(* IEC 61131-3 sources: com.logicals.lc3.webinar/RPMControl_Webinar/src_PRG_MQTT_RevPi_ST, 4 files *)

(* ---- PRG_RevPi_MQTTConnect.iecst ---- *)
/*
 * TauriL
 * MQTTConnect Task
 */

USING com.logicals.Basic.Logic;

PROGRAM PRG_RevPi_MQTTConnect

    VAR_EXTERNAL
      gstruc_MQTTClient    : DT_MQTTClient;
    END_VAR

    VAR_EXTERNAL
      /*
       * Funktion Publish starten (WebCon)
       */
       gx_MQTTPublish      : BOOL;
       gx_MQTTPublishState : BOOL;
    END_VAR

    VAR_EXTERNAL
       /*
        * Funktion Subscribe starten (WebCon)
        */
        gx_MQTTSubscribe      : BOOL;
        gx_MQTTSubscribeState : BOOL;
    END_VAR

   /*
    * PRG_RevPi_MQTTConnect
    */
	VAR_EXTERNAL
      /*
       * Globaler TraceLevel
       */
       gui_TraceLevel : UINT;
	END_VAR
   /*
    * Status Verbindung zum Broker
    */
	VAR_EXTERNAL
		/*
		 * State und Channel vom Connect
		 */
		 MQTT_State   : MQTT_SUBSCRIBER_STATE;
		 MQTT_Channel : DINT;
	END_VAR

    VAR_EXTERNAL
        /*
         * Conecting Status an WebCon
         */
         gui_MQTTConnecting    : UINT; // Anzahl der Zyklen in MQTTConnecting
        /*
         * Conect und DisConnect Status an WebCon
         */
	     gui_MQTTConOkCycle    : UINT; // Anzahl der Zyklen bis MQTT Connect
	     gui_MQTTConNotOkCycle : UINT; // Anzahl der Zyklen wenn MQTT DisConnect
        /*
         * Conect Status an WebCon
         */
         gx_MQTTConOk      : BOOL;
    END_VAR

    VAR

    l_ConState : MQTT_SUBSCRIBER_STATE;

    l_RC       : MQTT_RC;
    ldi_Ch     : DINT;

    l_RC_Disconnect : MQTT_RC;

  END_VAR

   VAR
    /*
     * DiagnoseBits fuer RTS
     */
     lx_RTSInit     : BOOL;
     lx_RTSRun      : BOOL;
     lx_RTSShutDown : BOOL;
     lx_RTSTerm     : BOOL;
   END_VAR

   VAR
	 //
	 // Aus HCLib
     // Alle Verbindungen bedienen
     // Hier werden die Daten konkret verschickt!
     FB_RevPi_MQTTConnect        : FB_MQTTConnect;
  END_VAR

 /*
  * Status MQTT Publish/Subscribe
  */
  VAR
     FB_Publish_Toogle         : FB_lc_Toggle_ST;
     FB_Subscribe_Toogle       : FB_lc_Toggle_ST;
  END_VAR

  VAR
    FB_MQTTCpyRevPiPar : FB_MQTTCpyRevPiPar;
  END_VAR

  VAR
    /*
     * Der Datentyp enthaelt alle wesentlichen Informationen f�r die Basis-
     * Einstellungen von MQTT
     */
     l_MQTTInitKom    : DT_MQTT;
  END_VAR

 /*
  * Initialisierungsmerker
  */
  VAR
     FB_InitR_TRIG       : R_TRIG;
  END_VAR

  VAR
    /* Lokaler InitPuls im Baustein */
     lx_CycleInit : BOOL;

    /* Lokaler Puls im Baustein */
     lx_CyclePulse : BOOL;
    /* Lokaler Zyklustaktzaehler */
     li_CycleCount : INT;

    /* Lokaler InitZyklustaktzaehler */
     li_CycleCountInitVal : INT;
  END_VAR

  VAR
    lstr_PRGName      : STRING[30] := 'PRG_RevPi_MQTTConnect';
    lui_TraceLevel    : UINT     := 5;

    lui_POU_UID       : UINT;                                      // Lokale POU-ID
    lstr_InstName     : STRING[30];
    lstr_POU_InstPath : STRING[128];                               // Lokale POU-ID
   END_VAR
 /*
  * -------------------------------------------------
  * Start SPS-Programm PRG_RevPi_MQTTConnect
  * -------------------------------------------------
  */
 /*
  * InitZyklus setzen wenn MQTT aktiv gesetzt!
  */
  FB_InitR_TRIG(CLK := TRUE,Q => lx_CycleInit);

 /*
  * CyclePulse
  */
  lx_CyclePulse := NOT(lx_CyclePulse);

 /*
  * LifeTick bzw. ZyklusZaehler
  */
  li_CycleCount := li_CycleCount + 1;

  IF lx_CycleInit = TRUE THEN
       /*
        * Globalen TraceLevel uebernehmen
        */
       lui_TraceLevel := gui_TraceLevel;
      /*
       * PI-Name fuer GVL-Liste
       */
       lstr_InstName        := GET_CURRENT_PI_NAME();
       lstr_POU_InstPath    := lstr_PRGName;
       li_CycleCountInitVal := li_CycleCountInitVal + 1;
   END_IF;

  /*
   * MQTT Parameter umkopieren
   */
   IF lx_CycleInit = TRUE THEN
    FB_MQTTCpyRevPiPar(vistruc_InitKom := l_MQTTInitKom,
                       vostruc_InitKom => gstruc_MQTTClient);
   END_IF;

   /*
    * Betriebsart MQTT von Visu
    * Publish der Daten immer aus TRUE im CycleInit setzen
    */
    FB_Publish_Toogle(vix_In := gx_MQTTPublish OR lx_CycleInit,vox_Out => gx_MQTTPublishState);
    FB_Subscribe_Toogle(vix_IN := gx_MQTTSubscribe, vox_Out =>gx_MQTTSubscribeState);

    /*
     * Es wird ein MQTT_Connect aufgebaut
     * Wird fuer Publish/Subscribe verwendet!
     * NUR ein Connect je Resource zum Broker erlaubt!
     *
     * Im RTSTerm bzw. RTSShutdown MUSS der Connect Disconnected werden!
     */
     FB_RevPi_MQTTConnect(vistr_InstPath                := lstr_InstName,
     	                  vistr_BrokerAddress          := l_MQTTInitKom.BrokerAdress,
                          vistr_ClientID               := l_MQTTInitKom.RevPiClientID,
                          vo_State                     => l_ConState,              // Status fuer Connect fuer alle zu oeffnenden Verbindungen (Pub/Sub) zum Broker
                          vo_RC                        => l_RC,                    // Status fuer Connect fuer alle zu oeffnenden Fehler (Pub/Sub) zum Broker
                          vodi_ch                      => ldi_Ch,                  // Status fuer Connect fuer alle zu oeffnenden Kanaele (Pub/Sub) zum Broker
                          voui_CycleCount_Connecting   => gui_MQTTConnecting,
                          voui_CycleCount_Connected    => gui_MQTTConOkCycle,      // Wert auch in WebCon
                          voui_CycleCount_NotConnected => gui_MQTTConNotOkCycle,   // Wert auch in WebCon
                          vox_MQTTConOk                => gx_MQTTConOk);           // Wert auch in WebCon

   gstruc_MQTTClient.x_MQTTConOk          := gx_MQTTConOk;
   gstruc_MQTTClient.ui_MQTTConnecting    := gui_MQTTConnecting;
   gstruc_MQTTClient.ui_MQTTConOkCycle    := gui_MQTTConOkCycle;
   gstruc_MQTTClient.ui_MQTTConNotOkCycle := gui_MQTTConNotOkCycle;

   /*
    * Ausgabe der Daten!
    */
    MQTT_State   := l_ConState;
    MQTT_Channel := ldi_ch;

   /*
    * Diagnosebits des RTS
    */
    RTSCycleInfo(Init     => lx_RTSInit,
  	             Run      => lx_RTSRun,
  	             Shutdown => lx_RTSShutDown,
  	             Term     => lx_RTSTerm);

   /*
    * Disconnect!
    * In RTS.CFG ShutDown Cycle von 3 Sekunden eintragen!
    */
    IF lx_RTSTerm = TRUE OR lx_RTSShutDown = TRUE THEN
     MQTT_Disconnect(ch := ldi_ch,
                     rc => l_RC_Disconnect);
     MQTT_State   := l_ConState;
     MQTT_Channel := -1;
    END_IF;

END_PROGRAM

(* ---- PRG_RevPi_MQTTPublish_Header.iecst ---- *)
 /*
  * logi.cals GmbH
  * A-3100 St. Poelten
  * Europaplatz 7/1
  * Tel.: 0043-5-77147
  *
  * logi.cals automation solutions & services GmbH
  * D-40738 Langenfeld
  * Postfach 1306
  * Tel.: 0043-5-77147
  *
  * Contact:
  * dieter.goltz@logicals.com
  *
  * History:
  * Created:
  * DG 2021-05-30 MQTT Header
  *
  * Modified:
  * DG 2021-05-30 MQTT Publish Header
  */

 /*
  * Description
  * ===========
  */

 /*
  * Beschreibung
  * ============
  * MQTT Kommunikation
  * Publish Header
  *
  */

/*
 * Lokaler Test
 * ============
 * sudo mosquitto_sub -d -t test   - test = Name des Topic -> /Tauri       - Header
 *                                                            /Tauri       - Werte
 *
 * sudo mosquitto_pub -d -t test –m “Hello” - test = Name des Topic -> /GHaus       - Header
 *                                                                     /GHaus/Value - Werte
 *
 *                               -m "Hello" -> String der verschickt wird!
 */

/*
 * Publish des Header von TauriL
 */
PROGRAM PRG_RevPi_MQTTPublish_Header
    /*
	 * PRG_RevPi_MQTTPublish_Header
	 */
    VAR_EXTERNAL
         MQTTHeader       : MQTTHeader;
    END_VAR

    VAR_EXTERNAL
        /*
         * Funktion Publish starten (WebCon)
         * Wird in MQTTConnect gesetzt!
         * Kann von hier mit gx_MQTTPublish getoggled werden!
         */
         gx_MQTTPublish      : BOOL;
         gx_MQTTPublishState : BOOL;
    END_VAR

	VAR_EXTERNAL
	   /*
		* State und Channel vom Connect
		*/
		MQTT_State   : MQTT_SUBSCRIBER_STATE;
		MQTT_Channel : DINT;
	END_VAR

	VAR_EXTERNAL
      /*
       * Globaler TraceLevel
       */
     gui_TraceLevel : UINT;
	END_VAR

	VAR_EXTERNAL
    /*
     * Uhrzeit und Daten von TimeBaustein abholen
     * und auf Globale Var in Byte schreiben
     * Fuer MQTT
     */
  	 gb_RTSSeconds : BYTE;
 	 gb_RTSMinutes : BYTE;
	 gb_RTSHours   : BYTE;

	 gb_RTSDay         : BYTE;
	 gb_RTSMonth       : BYTE;
	 gb_RTSYearHByte   : BYTE;
	 gb_RTSYearLByte   : BYTE;

    END_VAR

   VAR
      FB_MQTT_PublishRevPi      : FB_MQTT_Publish;
   END_VAR

  VAR
    /*
     * Der Datentyp enthaelt alle wesentlichen Initwerte f�r die MQTT-Kommunkation
     */
     l_MQTTInitKom         : DT_MQTT;
    /*
     * Status-Informationen
     */
     ldi_PublishLifeTick : DINT;
     lx_PublishOK        : BOOL;
     lui_IPVal1          : UINT;
     lui_IPVal2          : UINT;
     lui_IPVal3          : UINT;
     ldint_MQTTChannel   : DINT;
     ldint_MQTTCount     : DINT;
     ldint_MQTTrc        : DINT;
     lsint_MQTTState     : SINT;
     lx_MQTTENO          : BOOL;
     luint_MQTTLength    : UINT;
     lui_PubTick         : UINT;
  END_VAR

  VAR
    l_ConState : MQTT_SUBSCRIBER_STATE;
    ldi_ConCh  : DINT;
  END_VAR

  VAR
    lstr_PRGName   : STRING[30] := 'PRG_RevPi_MQTTPublish_Header';
    lui_TraceLevel : UINT     := 5;
  END_VAR

  VAR
     FB_InitR_TRIG       : R_TRIG;
  END_VAR

  VAR
    /* Lokaler InitPuls im Baustein */
     lx_CycleInit : BOOL;

    /* Lokaler Puls im Baustein */
     lx_CyclePulse : BOOL;
    /* Lokaler Zyklustaktzaehler */
     li_CycleCount : INT;

    /* Lokaler InitZyklustaktzaehler */
     li_CycleCountInitVal : INT;
  END_VAR

 /*
  * InitZyklus setzen wenn MQTT aktiv gesetzt!
  */
  FB_InitR_TRIG(CLK := TRUE,Q => lx_CycleInit);
 /*
  * CyclePulse
  */
  lx_CyclePulse := NOT(lx_CyclePulse);

 /*
  * LifeTick bzw. ZyklusZaehler
  */
  li_CycleCount := li_CycleCount + 1;

  /*
   * Steuerung Publish / Subscribe ueber die Visu
   *
   * Publish
   * Welche Daten sollen an den Broker zurueckgeschickt werden
   * Subscribe
   * Welche Daten sollen geholt werden?
   */
   IF lx_CycleInit = TRUE THEN
      /*
       * Init Messages senden
       */
       lui_TraceLevel := gui_TraceLevel;
       li_CycleCountInitVal := li_CycleCountInitVal + 1;
   END_IF;
   /*
    * Daten von MQTTConnect
    */
    l_ConState := MQTT_State;
    ldi_ConCh  := MQTT_Channel;

    IF l_ConState = MQTT_SUBSCRIBER_STATE#CONNECTED THEN

       IF gx_MQTTPublishState = TRUE THEN

     	 MQTTHeader.Second    := gb_RTSSeconds;
   	     MQTTHeader.Minute    := gb_RTSMinutes;
  	     MQTTHeader.Hour      := gb_RTSHours;

  	     MQTTHeader.Day       := gb_RTSDay;
  	     MQTTHeader.Month     := gb_RTSMonth;
  	     MQTTHeader.YearHByte := gb_RTSYearHByte;
  	     MQTTHeader.YearLByte := gb_RTSYearLByte;

         MQTTHeader.IPVal3 := TO_BYTE(RIGHT(IN:= l_MQTTInitKom.RevPiIPAdress, L := 1));
         MQTTHeader.IPVal2 := TO_BYTE(LEFT(RIGHT(IN:= l_MQTTInitKom.RevPiIPAdress, L := 2),1));
         MQTTHeader.IPVal1 := TO_BYTE(LEFT(RIGHT(IN:= l_MQTTInitKom.RevPiIPAdress, L := 3),1));

         FB_MQTT_PublishRevPi(vi_MQTTHeader            := MQTTHeader,
                              vistr_IPAddr             := l_MQTTInitKom.RevPiIPAdress,
                              vistr_BrokerIPAddr       := l_MQTTInitKom.BrokerAdress,
                              vix_Init                 := lx_CycleInit,
                              vi_State                 := l_ConState,
                              vdi_ch                   := ldi_ConCh,
         	                  vistr_BrokerPublishTopic := l_MQTTInitKom.RevPiTopic,
                              vodi_PublishLifeTick     => ldi_PublishLifeTick,
                              vox_PublishOK            => lx_PublishOK,
                              voui_IPVal1              => lui_IPVal1,
                              voui_IPVal2              => lui_IPVal2,
                              voui_IPVal3              => lui_IPVal3,
                              vodint_MQTTChannel       => ldint_MQTTChannel,
                              vodint_MQTTCount         => ldint_MQTTCount,
                              vodint_MQTTrc            => ldint_MQTTrc,
                              vosint_MQTTState         => lsint_MQTTState,
                              vox_MQTTENO              => lx_MQTTENO,
                              vouint_MQTTLength        => luint_MQTTLength,
                              voui_PubTick             => lui_PubTick);

        END_IF;
     END_IF;
END_PROGRAM

(* ---- PRG_RevPi_MQTTPublish_IO.iecst ---- *)
   /*
  * logi.cals GmbH
  * A-3100 St. Poelten
  * Europaplatz 7/1
  * Tel.: 0043-5-77147
  *
  * logi.cals automation solutions & services GmbH
  * D-40738 Langenfeld
  * Postfach 1306
  * Tel.: 0043-5-77147
  *
  * Contact:
  * dieter.goltz@logicals.com
  *
  * History:
  * Created:
  * DG 2021-05-30
  *
  * Modified:
  * DG 2021-05-30 IO
  */

 /*
  * Description
  * ===========
  */

 /*
  * Beschreibung
  * ============
  * MQTT Kommunikation
  * Publish Werte als Topics (IO)
  *
  * Austausch der aktuellen Daten mit dem Broker
  *
  */
 PROGRAM PRG_RevPi_MQTTPublish_IO

   VAR_EXTERNAL
        /*
         * Funktion Publish starten (WebCon)
         */
         gx_MQTTPublish      : BOOL;
         gx_MQTTPublishState : BOOL;
   END_VAR

   VAR_EXTERNAL
	    /* ProcessValue - Analogeingang_1 0..32767 unskaliert */
		gr_PV : REAL;
	    /* SetPoint     - Analogeingang_2 0..32767 unskaliert */
		gr_SP : REAL;
	    /* OutValue     - Analogausgang_1 0..32767 skaliert von 0..100% */
		gr_Y : REAL;
	    /* OutValue     - Ausgang Regler 0..100% wird skaliert auf 0..32767 */
		gr_PID_OUT : REAL;

	    /* ManualWert 0..100% */
		gr_Manual : REAL;

	    /* ProcessValue - Analogeingang_1 Skaliert 0..100%*/
		gr_PV_Scale : REAL;
	    /* SetPoint     - Analogeingang_2 Skaliert 0..100% */
		gr_SP_Scale : REAL;
	    /* OutValue     - Analogausgang_1 Skaliert 0..100% */
		gr_Y_Scale  : REAL;
        /*
         * Anzeige der Betriebsart 1Aus4
         */
        /* An Ausgang Ausgangswert = 0% */
        gx_ModeRPM0 : BOOL;
        /* An Ausgang Ausgangswert = 25% */
        gx_ModeRPM1 : BOOL;
        /* An Ausgang Ausgangswert = 50% */
        gx_ModeRPM2 : BOOL;
        /* An Ausgang SetPoint von Poti */
        gx_ModeRPM3 : BOOL;
        /* An Ausgang SetPoint von SFC */
        gx_ModeRPM4 : BOOL;

        /* Blinkfunktion */
        gx_Flash : BOOL;
   END_VAR
  /*
   * PRG_TauriL_MQTTPublish_IO
   */
   VAR_EXTERNAL
    /*
     * State und Channel vom Connect
     */
     MQTT_State   : MQTT_SUBSCRIBER_STATE;
     MQTT_Channel : DINT;
   END_VAR

   VAR_EXTERNAL
      /*
       * Globaler TraceLevel
       */
       gui_TraceLevel : UINT;
   END_VAR

  /*
   * Publish Topic / BOOL-Status von Topic
   */
   VAR
       FB_MQTT_Publish_IOBlink             : FB_MQTT_Publish_IO;

       FB_MQTT_Publish_IOValModeRPM0       : FB_MQTT_Publish_IO;
       FB_MQTT_Publish_IOValModeRPM1       : FB_MQTT_Publish_IO;
       FB_MQTT_Publish_IOValModeRPM2       : FB_MQTT_Publish_IO;
       FB_MQTT_Publish_IOValModeRPM3       : FB_MQTT_Publish_IO;
       FB_MQTT_Publish_IOValModeRPM4       : FB_MQTT_Publish_IO;

       FB_MQTT_Publish_IOValPV             : FB_MQTT_Publish_IOVal;
       FB_MQTT_Publish_IOValSP             : FB_MQTT_Publish_IOVal;
       FB_MQTT_Publish_IOValY              : FB_MQTT_Publish_IOVal;
       FB_MQTT_Publish_IOValManual         : FB_MQTT_Publish_IOVal;
       FB_MQTT_Publish_IOValPV_Scale       : FB_MQTT_Publish_IOVal;
       FB_MQTT_Publish_IOValSP_Scale       : FB_MQTT_Publish_IOVal;
       FB_MQTT_Publish_IOValY_Scale        : FB_MQTT_Publish_IOVal;

   END_VAR

  VAR
    /*
     * Der Datentyp enthaelt alle wesentlichen Informationen fuer die Basis-
     * Einstellungen von MQTT
     */
     l_MQTTInitKom    : DT_MQTT;
  END_VAR

  VAR
    l_ConState : MQTT_SUBSCRIBER_STATE;
    ldi_ConCh  : DINT;
  END_VAR

   VAR
    lstr_PRGName : STRING[30] := 'PRG_TauriL_MQTTPublish_IO';
    lui_TraceLevel : UINT     := 5;
   END_VAR
 /*
  * Initialisierungsmerker
  */
  VAR
     FB_InitR_TRIG       : R_TRIG;
  END_VAR

  VAR
    /* Lokaler InitPuls im Baustein */
     lx_CycleInit        : BOOL;

    /* Lokaler Puls im Baustein */
     lx_CyclePulse       : BOOL;
    /* Lokaler Zyklustaktzaehler */
     li_CycleCount       : INT;

    /* Lokaler InitZyklustaktzaehler */
     li_CycleCountInitVal : INT;
  END_VAR

  /*
   * InitZyklus setzen wenn MQTT aktiv gesetzt!
   */
   FB_InitR_TRIG(CLK := TRUE,Q => lx_CycleInit);

   lui_TraceLevel := gui_TraceLevel;

  /*
   * CyclePulse
   */
   lx_CyclePulse := NOT(lx_CyclePulse);

  /*
   * LifeTick bzw. ZyklusZaehler
   */
   li_CycleCount := li_CycleCount + 1;
  /*
   * -------------------------------------------------
   * Start SPS-Programm PRG_TauriL_MQTTPublish_IO
   * -------------------------------------------------
   */

  /*
   * Steuerung Publish_IO
   *
   * Publish
   * Welche Einzel-Daten sollen an den Broker geschickt werden
   */
   IF lx_CycleInit = TRUE THEN
       li_CycleCountInitVal := li_CycleCountInitVal + 1;
   END_IF;

   /*
    * Daten von MQTTConnect
    */
    l_ConState := MQTT_State;
    ldi_ConCh  := MQTT_Channel;

   /*
    * Kommt von MQTTConnect
    * Wert MUSS 6 sein!
    */
    IF l_ConState = MQTT_SUBSCRIBER_STATE#CONNECTED /* connected */ THEN

      IF gx_MQTTPublishState = TRUE THEN

      /*
       * Blinkfunktion an gx_Out8
       */
       FB_MQTT_Publish_IOBlink(viui_TraceLevel            := lui_TraceLevel,
                               vix_PubIn                  := gx_Flash,
                               vistr_BrokerPublishTopicIO := l_MQTTInitKom.TauriLTopicIOBlink,
                               vi_State                   := l_ConState,
                               vidi_Ch                    := ldi_ConCh);

      /*
       * Mode RPM 0
       */
       FB_MQTT_Publish_IOValModeRPM0(viui_TraceLevel            := lui_TraceLevel,
                                     vix_PubIn                  := gx_ModeRPM0,
                                     vistr_BrokerPublishTopicIO := l_MQTTInitKom.TauriLTopicIOModeRPM0,
                                     vi_State                   := l_ConState,
                                     vidi_Ch                    := ldi_ConCh);

      /*
       * Mode RPM 1
       */
       FB_MQTT_Publish_IOValModeRPM1(viui_TraceLevel            := lui_TraceLevel,
                                     vix_PubIn                  := gx_ModeRPM1,
                                     vistr_BrokerPublishTopicIO := l_MQTTInitKom.TauriLTopicIOModeRPM1,
                                     vi_State                   := l_ConState,
                                     vidi_Ch                    := ldi_ConCh);

      /*
       * Mode RPM 2
       */
       FB_MQTT_Publish_IOValModeRPM2(viui_TraceLevel            := lui_TraceLevel,
                                     vix_PubIn                  := gx_ModeRPM2,
                                     vistr_BrokerPublishTopicIO := l_MQTTInitKom.TauriLTopicIOModeRPM2,
                                     vi_State                   := l_ConState,
                                     vidi_Ch                    := ldi_ConCh);

      /*
       * Mode RPM 3
       */
       FB_MQTT_Publish_IOValModeRPM3(viui_TraceLevel            := lui_TraceLevel,
                                     vix_PubIn                  := gx_ModeRPM3,
                                     vistr_BrokerPublishTopicIO := l_MQTTInitKom.TauriLTopicIOModeRPM3,
                                     vi_State                   := l_ConState,
                                     vidi_Ch                    := ldi_ConCh);
      /*
       * Mode RPM 4
       */
       FB_MQTT_Publish_IOValModeRPM4(viui_TraceLevel            := lui_TraceLevel,
                                     vix_PubIn                  := gx_ModeRPM4,
                                     vistr_BrokerPublishTopicIO := l_MQTTInitKom.TauriLTopicIOModeRPM4,
                                     vi_State                   := l_ConState,
                                     vidi_Ch                    := ldi_ConCh);
      /*
       * PV
       */
       FB_MQTT_Publish_IOValPV(viui_TraceLevel            := lui_TraceLevel,
                               vir_PubIn                  := gr_PV,
                               vistr_BrokerPublishTopicIO := l_MQTTInitKom.TauriLTopicIOPV,
                               vi_State                   := l_ConState,
                               vidi_Ch                    := ldi_ConCh);

      /*
       * SP
       */
       FB_MQTT_Publish_IOValSP(viui_TraceLevel            := lui_TraceLevel,
                               vir_PubIn                  := gr_SP,
                               vistr_BrokerPublishTopicIO := l_MQTTInitKom.TauriLTopicIOSP,
                               vi_State                   := l_ConState,
                               vidi_Ch                    := ldi_ConCh);

      /*
       * Y
       */
       FB_MQTT_Publish_IOValY(viui_TraceLevel            := lui_TraceLevel,
                               vir_PubIn                  := gr_Y,
                               vistr_BrokerPublishTopicIO := l_MQTTInitKom.TauriLTopicIOY,
                               vi_State                   := l_ConState,
                               vidi_Ch                    := ldi_ConCh);

      /*
       * PV_Scale
       */
       FB_MQTT_Publish_IOValPV_Scale(viui_TraceLevel            := lui_TraceLevel,
                                     vir_PubIn                  := gr_PV_Scale,
                                     vistr_BrokerPublishTopicIO := l_MQTTInitKom.TauriLTopicIOPV_Scale,
                                     vi_State                   := l_ConState,
                                     vidi_Ch                    := ldi_ConCh);

      /*
       * SP_Scale
       */
       FB_MQTT_Publish_IOValSP_Scale(viui_TraceLevel            := lui_TraceLevel,
                                     vir_PubIn                  := gr_SP_Scale,
                                     vistr_BrokerPublishTopicIO := l_MQTTInitKom.TauriLTopicIOSP_Scale,
                                     vi_State                   := l_ConState,
                                     vidi_Ch                    := ldi_ConCh);

      /*
       * Y = PID_OUT = Stellsignale des Reglers OHNE Skalierung 0..100%
       */
       FB_MQTT_Publish_IOValY_Scale(viui_TraceLevel            := lui_TraceLevel,
                                    vir_PubIn                  := gr_Y_Scale,
                                    vistr_BrokerPublishTopicIO := l_MQTTInitKom.TauriLTopicIOY_Scale,
                                    vi_State                   := l_ConState,
                                    vidi_Ch                    := ldi_ConCh);
   //
   //   /*
   //    * Manual
   //    */
   //    FB_MQTT_Publish_IOValManual(viui_TraceLevel            := lui_TraceLevel,
   //                                 vir_PubIn                  := gr_Manual,
   //                                 vistr_BrokerPublishTopicIO := l_MQTTInitKom.TauriTopicIOManual,
   //                                 vi_State                   := l_ConState,
   //                                 vidi_Ch                    := ldi_ConCh);
   //
      END_IF;
   END_IF;

  END_PROGRAM

(* ---- PRG_RevPi_MQTTSubscribe_Header.iecst ---- *)
 /*
  * logi.cals GmbH
  * A-3100 St. Poelten
  * Europaplatz 7/1
  * Tel.: 0043-5-77147
  *
  * logi.cals automation solutions & services GmbH
  * D-40738 Langenfeld
  * Postfach 1306
  * Tel.: 0043-5-77147
  *
  * Contact:
  * dieter.goltz@logicals.com
  *
  * History:
  * Created:
  * DG 2021-04-04
  *
  * Modified:
  * DG 2021-02-28 - Anzahl Topics > 16 klaeren
  * DG 2021-04-11 - logi.Lib 0.0.4
  * DG 2021-09-05 - logi.Lib 0.0.17
  * DG 2021-09-20 - logi.Lib 0.0.20-SNAPSHOT
  *
  */

 /*
  * Description
  */

 /*
  * Beschreibung
  * MQTT-Kommunikation
  *
  */
USING com.logicals.Basic.Convert;
USING com.logicals.Basic.Trace;

/*
 * Subscribe Daten vom Broker holen
 */
PROGRAM PRG_RevPi_MQTTSubscribe

	VAR_EXTERNAL
      /*
       * Globaler TraceLevel
       */
       gui_TraceLevel : UINT;
	END_VAR

    VAR_EXTERNAL
         MQTTHeader       : MQTTHeader;
    END_VAR

	VAR_EXTERNAL
		/*
		 * State und Channel vom Connect
		 */
		 MQTT_State   : MQTT_SUBSCRIBER_STATE;
		 MQTT_Channel : DINT;
	END_VAR

    VAR
      lui_TaskID      : UINT;
      lstr_TaskName   : STRING[50];

      lui_TaskSetTime : UINT;
      lui_TaskActTime : UINT;
    END_VAR

    VAR
      l_ConState : MQTT_SUBSCRIBER_STATE;
      ldi_Ch     : DINT;
    END_VAR

    VAR
    /*
     * Diese Daten sollen als Array "Published" werden
     */
     larr_MQTT   : ARRAY [0..7] OF BYTE;    // Uebergabe des MQTT Array
     ldi_MQTTLen : DINT := 8;               // Laenge
    END_VAR

    VAR
	   /*
        * Der Datentyp enthaelt alle wesentlichen Initwerte fuer die MQTT-Kommunkation
        */
        l_MQTTInitKom  : DT_MQTT;
    END_VAR

    VAR
      /*
       * Raspi2
       */
       lx_Raspi2TopicOk1  : BOOL;
       lstr_Raspi2Topic1   : STRING[1024];
      /*
       * Raspi4
       */
       lx_Raspi4TopicOk1  : BOOL;
       lstr_Raspi4Topic1   : STRING[1024];
      /*
       * RevPi
       */
       lx_RevPiTopicOk1  : BOOL;
       lstr_RevPiTopic1   : STRING[1024];
      /*
       * TauriL
       */
       lx_TauriLTopicOk1  : BOOL;
       lstr_TauriLTopic1   : STRING[1024];

    END_VAR

	VAR
		larr_ioImageRemote    : ARRAY [0..1023] OF BYTE;
		ldi_ioImageRemoteSize : DINT := 1024;
		ldi_ioImageRemoteLen  : DINT := -1;

		lstr_ReceiveTopic      : STRING[255];

		larr_bImageRemote      : ARRAY [0..1023] OF BYTE;

	   /*
	    * Alle erhaltenen Topics
	    */
		lstrarr_TopicArray : ARRAY [MQTT_MsgBound#Min..MQTT_MsgBound#Max] OF STRING[255];

	   /*
	    * Alle erhaltenen RC-Werte
	    */
		ldiarr_MessageRC : ARRAY [MQTT_MsgBound#Min..MQTT_MsgBound#Max] OF DINT;

	   /*
	    * Alle erhaltenen MessageLen-Werte
	    */
		ldiarr_MessageLen : ARRAY [MQTT_MsgBound#Min..MQTT_MsgBound#Max] OF DINT;

       /*
        * Raspi2
        */
		lui_Raspi2MessageLength1    : UINT;

       /*
        * Raspi4
        */
		lui_Raspi4MessageLength1    : UINT;

       /*
        * RevPi
        */
		lui_RevPiMessageLength1   : UINT;

       /*
        * TauriL
        */
		lui_TauriLMessageLength1    : UINT;

       /*
        * MessageLifeTick
        */
       /*
        * Raspi2
        */
		lui_Raspi2MessageLifeTick1  : UINT;

       /*
        * Raspi4
        */
		lui_Raspi4MessageLifeTick1  : UINT;

       /*
        * RevPi
        */
		lui_RevPiMessageLifeTick1  : UINT;

       /*
        * TauriL
        */
		lui_TauriLMessageLifeTick1  : UINT;

       /*
        * MessageRC
        */
       /*
        * Raspi2
        */
		ldi_Raspi2MessageRC1   : DINT;
       /*
        * Raspi4
        */
		ldi_Raspi4MessageRC1   : DINT;

       /*
        * RevPi
        */
		ldi_RevPiMessageRC1   : DINT;

       /*
        * TauriL
        */
		ldi_TauriLMessageRC1   : DINT;
       /*
        * MessagePos
        */
       /*
        * Raspi2
        */
		lui_Raspi2MessagePosIdx1   : UINT;

       /*
        * Raspi4
        */
		lui_Raspi4MessagePosIdx1   : UINT;

       /*
        * RevPi
        */
		lui_RevPiMessagePosIdx1    : UINT;

       /*
        * TauriL
        */
		lui_TauriLMessagePosIdx1   : UINT;

	   /*
	    * Subscribe-Flags von RevPi
	    */
	    lx_CL1_subscribed   : BOOL := FALSE;  //
	    lx_CL2_subscribed   : BOOL := FALSE;  //
		lx_CL3_subscribed   : BOOL := FALSE;  //
		lx_CL4_subscribed   : BOOL := FALSE;  //
		lx_CL5_subscribed   : BOOL := FALSE;  //
		lx_CL6_subscribed   : BOOL := FALSE;  //
		lx_CL7_subscribed   : BOOL := FALSE;  //
		lx_CL8_subscribed   : BOOL := FALSE;  //
		lx_CL9_subscribed   : BOOL := FALSE;  //
		lx_CL10_subscribed  : BOOL := FALSE;  //

		message_received : BOOL := FALSE;

		lrc_ReceiveTopic : MQTT_RC;

       /*
        * RC fuer Subscribe vom RevPi
        */
		rc_CL1  : MQTT_RC;
		rc_CL2  : MQTT_RC;
		rc_CL3  : MQTT_RC;
		rc_CL4  : MQTT_RC;
		rc_CL5  : MQTT_RC;
		rc_CL6  : MQTT_RC;
		rc_CL7  : MQTT_RC;
		rc_CL8  : MQTT_RC;
		rc_CL9  : MQTT_RC;
		rc_CL10 : MQTT_RC;

       /*
        * Puffer fuer Empfangsdaten
        */
		lstrarr_Messages     : ARRAY [MQTT_MsgBound#Min..MQTT_MsgBound#Max] OF STRING[1024];

		lusi_MessageIndex    : USINT := 0;
		lusi_MessageIndexMin : USINT := MQTT_MsgBound#Min;
		lusi_MessageIndexMax : USINT := MQTT_MsgBound#Max;

	END_VAR

    VAR
      FB_HCTrace        : FB_lc_Trace_ST;
      lstr_PRGName      : STRING[30] := 'PRG_RevPi_MQTTSubscribe_Header';
      lstr_InstName     : STRING[30];
      lui_TraceLevel    : UINT       := 5;
      lstr_POU_InstPath : STRING[128];                               // Lokale POU-ID
    END_VAR

    VAR
      FB_InitR_TRIG       : R_TRIG;
    END_VAR

	VAR
	  li_CycleCount : INT;
	  lx_CycleInit  : BOOL;
	  lx_CyclePulse : BOOL;
      li_CycleCountInitVal : INT;
	END_VAR

	FB_InitR_TRIG(CLK := TRUE, Q => lx_CycleInit);

   /*
    * Laesst die Moeglichkeit zu den TraceLevel lokal zu aendern!
    */
    IF lx_CycleInit = TRUE THEN
	   lui_TraceLevel       := gui_TraceLevel;
       lstr_InstName        := GET_CURRENT_PI_NAME();
       lstr_POU_InstPath    := lstr_InstName;
       li_CycleCountInitVal := li_CycleCountInitVal + 1;
       FB_HCTrace (vistr_TraceText := CONCAT(IN1 := lstr_PRGName, IN2 := ' Init'), viui_TraceLevel := lui_TraceLevel);
	END_IF;

	li_CycleCount := li_CycleCount + 1;
	lx_CyclePulse := NOT lx_CyclePulse;
   /*
    * Status abfragen ueber das IOSubSystem MQTT des RTS
    */
//	MQTT_State := MQTT_GetState(ch := ldi_Ch, rc => rc, ENO => ENO);

   /*
    * Interne Werte mit Uebergabe von MQTTConnect!
    */
    l_ConState := MQTT_State;
    ldi_ch     := MQTT_Channel;

   /*
    * Uebergabe State von MQTTConnect!
    */
	IF l_ConState = MQTT_SUBSCRIBER_STATE#CONNECTED THEN

		/* connect to topic in case connection has been established */
		IF NOT(lx_CL1_subscribed) THEN
            /* Topics von Raspi2 */
            MQTT_Subscribe(ch := ldi_Ch, topic := l_MQTTInitKom.Raspi2Topic,                rc => rc_CL1); // '/Server', rc => rc_CL1);

			lx_CL1_subscribed := rc_CL1 = MQTT_RC#OK;
        END_IF;

		IF NOT(lx_CL2_subscribed) THEN
//          /* Topics von Raspi4 */
			MQTT_Subscribe(ch := ldi_Ch, topic := l_MQTTInitKom.Raspi4Topic,                 rc => rc_CL2); //

			lx_CL2_subscribed := rc_CL2 = MQTT_RC#OK;
        END_IF;

		IF NOT(lx_CL3_subscribed) THEN
//          /* Topics von RevPi */
 			MQTT_Subscribe(ch := ldi_Ch, topic := l_MQTTInitKom.RevPiTopic, rc => rc_CL3);

			lx_CL3_subscribed := rc_CL3 = MQTT_RC#OK;
        END_IF;

		IF NOT(lx_CL4_subscribed) THEN
//          /* Topics von TauriL */
           MQTT_Subscribe(ch := ldi_Ch, topic := l_MQTTInitKom.TauriLTopic, rc => rc_CL4);

			lx_CL4_subscribed := rc_CL4 = MQTT_RC#OK;
        END_IF;

		IF NOT(lx_CL5_subscribed) THEN

			lx_CL5_subscribed := rc_CL5 = MQTT_RC#OK;
        END_IF;

		IF NOT(lx_CL6_subscribed) THEN

			lx_CL6_subscribed := rc_CL6 = MQTT_RC#OK;
        END_IF;

		IF NOT(lx_CL7_subscribed) THEN

			lx_CL7_subscribed := rc_CL7 = MQTT_RC#OK;
        END_IF;

		IF NOT(lx_CL8_subscribed) THEN
//          /*  */

			lx_CL8_subscribed := rc_CL8 = MQTT_RC#OK;
        END_IF;

		IF NOT(lx_CL9_subscribed) THEN
//          /*  */

			lx_CL9_subscribed := rc_CL9 = MQTT_RC#OK;
        END_IF;

		IF NOT(lx_CL10_subscribed) THEN
//          /*  */

			lx_CL10_subscribed := rc_CL10 = MQTT_RC#OK;
        END_IF;

 //    MQTT_RC : DINT(OK := 0,
 //                  ERROR := 1,
 //                  ERROR_MEM_ALLOC := 2,
 //                  ERROR_CONNECT := 3,
 //                  ERROR_CH_INVALID := 4,
 //                  ERROR_OUT_OF_CLIENTS := 5,
 //                  ERROR_OUT_OF_CB := 6,
 //                  ERROR_INVALID_MUTEX := 7,
 //                  ERROR_NO_MSG_RECEIVED := 8,
 //                  ERROR_NO_MSG_PUBLISHED := 9,
 //                  ERROR_MSG_TRUNCATED := 10,
 //                  ERROR_CH_INVALID_STATE := 11,
 //                  ERROR_CANNOT_DISCONNECT := 12,
 //                  ERROR_AUTHENTICATION_FAILED := 13,
 //                  ERROR_SSL_NOT_SUPPORTED := 14);

	   /*
		* clear the receive ring buffer
		*/
		FOR lusi_MessageIndex := MQTT_MsgBound#Min TO MQTT_MsgBound#Max DO // 0 TO 20 DO
		  lstrarr_Messages[lusi_MessageIndex] := '';
		END_FOR;

		/*
		 * if subscribed, obtain only the latest message
		 */
		message_received := FALSE;
		lusi_MessageIndex    := 0;

		REPEAT
			lstr_ReceiveTopic := MQTT_Receive(ch          := ldi_Ch,
				                              payload     := REF(larr_ioImageRemote[0]),
				                              payload_len := ldi_ioImageRemoteSize,
				                              len         => ldi_ioImageRemoteLen,
				                              rc          => lrc_ReceiveTopic);

			message_received := TRUE;

			// convert the received byte array to a string
			lstrarr_Messages[lusi_MessageIndex] := FUN_lc_StrFromByteArr_C(larr_ioImageRemote, ldi_ioImageRemoteLen);
           /*
            * Das erhaltene Topic im Array hinterlegen
            */
            lstrarr_TopicArray[lusi_MessageIndex] := lstr_ReceiveTopic;
            ldiarr_MessageRC[lusi_MessageIndex]   := lrc_ReceiveTopic;
            ldiarr_MessageLen[lusi_MessageIndex]  := ldi_ioImageRemoteLen;

			//
			// Messages-Index anpassen fuer weitere Nachrichten
			if (lusi_MessageIndex < lusi_MessageIndexMax) THEN
				lusi_MessageIndex := lusi_MessageIndex + 1;
			ELSE
				lusi_MessageIndex := lusi_MessageIndexMin;
                FB_HCTrace (vistr_TraceText := CONCAT(IN1 := lstr_PRGName, IN2 := 'WARNING: MQTT message buffer overrun!'), viui_TraceLevel := lui_TraceLevel);
			END_IF;

			IF lrc_ReceiveTopic <> MQTT_RC#OK THEN
                FB_HCTrace (vistr_TraceText := CONCAT(IN1 := lstr_PRGName, IN2 := ' rc <> MQTT_RC#OK := ', IN3 := TO_STRING(lrc_ReceiveTopic)), viui_TraceLevel := lui_TraceLevel);
				EXIT;
			ELSE
                FB_HCTrace (vistr_TraceText := CONCAT(IN1 := lstr_PRGName, IN2 := ' Message received: Topic := ', IN3 := lstr_ReceiveTopic), viui_TraceLevel := lui_TraceLevel);
			END_IF;

		UNTIL FALSE

		END_REPEAT;
	END_IF;

    lx_Raspi2TopicOk1    := FALSE;
    lx_Raspi4TopicOk1    := FALSE;
    lx_RevPiTopicOk1     := FALSE;
    lx_TauriLTopicOk1    := FALSE;

   /*
    * Das Array der empfangenen Topics fuer Server analysieren
    */
    FOR lusi_MessageIndex := MQTT_MsgBound#Min TO MQTT_MsgBound#Max DO // 0 TO 20 DO

    /*
     * Header Raspi2
     */
     IF lstrarr_TopicArray[lusi_MessageIndex] = l_MQTTInitKom.Raspi2Topic AND lx_Raspi2TopicOk1 = FALSE THEN
       lui_Raspi2MessagePosIdx1   := lusi_MessageIndex;
       lui_Raspi2MessageLifeTick1 := lui_Raspi2MessageLifeTick1 + 1;
       lui_Raspi2MessageLength1   := TO_UINT(ldiarr_MessageLen[lusi_MessageIndex]);
       ldi_Raspi2MessageRC1       := ldiarr_MessageRC[lusi_MessageIndex];
        lx_Raspi2TopicOk1         := TRUE;

       larr_bImageRemote := FUN_lc_ByteArrFromStr_C(vistr_Arr := lstrarr_Messages[lusi_MessageIndex], vidi_len := ldiarr_MessageLen[lusi_MessageIndex]);

       lstr_Raspi2Topic1 := lstrarr_Messages[lusi_MessageIndex];
     END_IF;

    /*
     * Header Raspi4
     */
     IF lstrarr_TopicArray[lusi_MessageIndex] = l_MQTTInitKom.Raspi4Topic AND lx_Raspi4TopicOk1 = FALSE THEN
       lui_Raspi4MessagePosIdx1   := lusi_MessageIndex;
       lui_Raspi4MessageLifeTick1 := lui_Raspi4MessageLifeTick1 + 1;
       lui_Raspi4MessageLength1   := TO_UINT(ldiarr_MessageLen[lusi_MessageIndex]); // len(lstrarr_Messages[lusi_MessageIndex]);
       ldi_Raspi4MessageRC1       := ldiarr_MessageRC[lusi_MessageIndex];
       lx_Raspi4TopicOk1          := TRUE;

       larr_bImageRemote := FUN_lc_ByteArrFromStr_C(vistr_Arr := lstrarr_Messages[lusi_MessageIndex], vidi_len := ldiarr_MessageLen[lusi_MessageIndex]);

       lstr_Raspi4Topic1 := lstrarr_Messages[lusi_MessageIndex];

     END_IF;

    /*
     * Header RevPi
     */
     IF lstrarr_TopicArray[lusi_MessageIndex] = l_MQTTInitKom.RevPiTopic AND lx_RevPiTopicOk1 = FALSE THEN // '/RevPi_IO/HellMld' THEN
       lui_RevPiMessagePosIdx1   := lusi_MessageIndex;
       lui_RevPiMessageLifeTick1 := lui_RevPiMessageLifeTick1 + 1;
       lui_RevPiMessageLength1   := TO_UINT(ldiarr_MessageLen[lusi_MessageIndex]); // len(lstrarr_Messages[lusi_MessageIndex]);
       ldi_RevPiMessageRC1       := ldiarr_MessageRC[lusi_MessageIndex];
       lx_RevPiTopicOk1          := TRUE;

       larr_bImageRemote := FUN_lc_ByteArrFromStr_C(vistr_Arr := lstrarr_Messages[lusi_MessageIndex], vidi_len := ldiarr_MessageLen[lusi_MessageIndex]);

       lstr_RevPiTopic1 := lstrarr_Messages[lusi_MessageIndex];

     END_IF;

    /*
     * Header TauriL
     */
     IF lstrarr_TopicArray[lusi_MessageIndex] = l_MQTTInitKom.TauriLTopic AND lx_TauriLTopicOk1 = FALSE THEN // '/TauriL_IO/HellMld' THEN
       lui_TauriLMessagePosIdx1   := lusi_MessageIndex;
       lui_TauriLMessageLifeTick1 := lui_TauriLMessageLifeTick1 + 1;
       lui_TauriLMessageLength1   := TO_UINT(ldiarr_MessageLen[lusi_MessageIndex]); // len(lstrarr_Messages[lusi_MessageIndex]);
       ldi_TauriLMessageRC1       := ldiarr_MessageRC[lusi_MessageIndex];
       lx_TauriLTopicOk1          := TRUE;

       lstr_TauriLTopic1 := lstrarr_Messages[lusi_MessageIndex];

     END_IF;

    /*
     * Alle gefunden!
     */
     IF lx_Raspi2TopicOk1 = TRUE AND lx_Raspi4TopicOk1  = TRUE AND lx_RevPiTopicOk1  = TRUE AND lx_TauriLTopicOk1  = TRUE THEN
       lusi_MessageIndex := MQTT_MsgBound#Max;
     END_IF;

    END_FOR;

END_PROGRAM
